PROGRAM MAIN
VAR
END_VAR

END_PROGRAM

(* stored: Version 1.1.0.1
   POU MAIN: Id {13aa0b6a-1832-4149-b405-c6ea458a212e} *)
